{attribute 'pack_mode' := '1'}
TYPE ST_1001_Initialize_position :
	STRUCT
		Header : ST_SupervisorHeader := (nMessageID := 1001, nMessageLength := 24);
		X	   : REAL; //		X - map coordinate OF the AGV in meters
		Y	   : REAL; //		Y - map coordinate of the AGV in meters
		H	   : REAL; //		Heading of the AGV on the map in radians
		Level  : DINT; //	The level ID on which the AGV is located
	END_STRUCT
END_TYPE

(* stored: Version 1.1.0.1, ProductVersion 3.1.4026.17
   DUT ST_1001_Initialize_position: Id {bc9f0d1c-ab16-4cd1-be97-b6a9753db434} *)
